INTERFACE I_ArrayDatatype EXTENDS I_UserDefinedDatatype

METHOD PUBLIC ABSTRACT GetElementAsDatatypeByIndex : I_Datatype
VAR_INPUT
	Index : DINT;
END_VAR
END_METHOD

PROPERTY PUBLIC ABSTRACT LowerBound : DINT
GET
END_GET
END_PROPERTY

PROPERTY PUBLIC ABSTRACT UpperBound : DINT
GET
END_GET
END_PROPERTY

END_INTERFACE

(* stored: Version 1.1.0.1, ProductVersion 3.1.4024.13
   Itf I_ArrayDatatype: Id {a8e57a5b-bfda-0173-132d-0647d5e8567e}
   Method GetElementAsDatatypeByIndex: Id {973559c5-0f11-0686-04fe-e501bbe80023}
   Property LowerBound: Id {c1062beb-c4a3-003a-39cf-c3c367a6b714}
   Get Get: Id {78acf8a9-4ffe-0e40-2dc2-422f83f59daf}
   Property UpperBound: Id {5ae63db9-c190-0d5f-0ab8-5e27de73fc4c}
   Get Get: Id {b47b1dac-3851-0071-0198-64b6048be994} *)
